// Mitsubishi GX Works2 project: b06   PLC: Q02/Q02H

PROGRAM MAIN
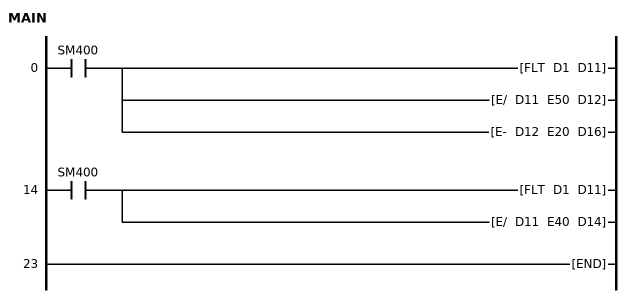
0     LD      SM400
      FLT     D1 D11
      E/      D11 E50 D12
      E-      D12 E20 D16
14    LD      SM400
      FLT     D1 D11
      E/      D11 E40 D14
23    END
END_PROGRAM
